FUNCTION_BLOCK FB_TopMold_OLD
VAR CONSTANT
	sCycleStateTextDef: ARRAY[0..25]  OF STRING :=	
		['State 0: Wait for Start',
		'State 1: Wait for signal to start move down',
		'State 2: Move down',
		'State 3: Drying lock time, Building pressure',
		'State 4: Start drying time',
		'State 5: Open pressure relief valve',
		'State 6: Vacuum time closed',
		'State 7: Move up',
		'State 8: Wait until take out unit is moving up and start blowoff',
		'State 9: Await blowoff time and stop blowoff',
		'State 10:',
		'State 11:',
		'State 12:',
		'State 13:',
		'State 14:',
		'State 15:',
		'State 16:',
		'State 17:',
		'State 18:',
		'State 19:',
		'State 20: Stop cycle state',																
		'State 21: Stop cycle state',
		'State 22:',
		'State 23:',
		'State 24:',
		'State 25:Stop direct state'];
	
	tCycleStateTimeouts: ARRAY[0..10] OF TIME := 
		[T#10S,T#10S,T#10S,T#10S,T#10S,T#10S,T#10S,T#10S,T#10S,T#10S,
		T#10S];

	sInitStateTextDef: ARRAY[0..10] OF STRING :=
		['State 0: Wait for Init Start',
		'State 1: Await pressure relief',
		'State 2: Move up',
		'State 3: Description Init State 3',
		'State 4: Description Init State 4',
		'State 5: Description Init State 5',
		'State 6: Description Init State 6',
		'State 7: Description Init State 7',
		'State 8: Description Init State 8',
		'State 9: Description Init State 9',
		'State 10: Stop init state'];

	tInitStateTimeouts: ARRAY[0..10] OF TIME := 
		[T#10S,T#10S,T#10S,T#10S,T#10S,T#10S,T#10S,T#10S,T#10S,T#10S
		,T#10S];
END_VAR

VAR_INPUT
	mxReset							: BOOL;	(*Reset Error*)
	mxEmergency						: BOOL;
	mxAutoMode						: BOOL; (* TRUE = Automode *)
	mxEmptyMachine					: BOOL;
	mxEnableHeating					: BOOL;

	mxResetCycleState				: BOOL;
	mxResetInitState				: BOOL;
	mxForceInit						: BOOL; (*Reset Calibration Flag*)

	mxMoveDown						: BOOL; (* Signal from bottommold *)
	mxMoveUp						: BOOL; (* Drying finished or transfer ready with new product *)
	mxTakeOutIsMovingUp: BOOL;
	RHSR_Blocked 					: BOOL;
END_VAR
VAR_IN_OUT
	MachParameters					: ST_TopMoldMachPar;
	ProdParameters					: ST_TopMoldProdPar;
END_VAR
VAR_OUTPUT
(*Errors*)
	Errors							: ST_TopMoldErrors;
	mxErrorInit						: BOOL;		(* Error, stop immediately. Initialisation neccesary *)
	mxErrorStopinPos				: BOOL;		(* Error, stop in position. Only reset neccesary *)

(* State vars *)
	mxCycleBusy						: BOOL;
	mxInitBusy						: BOOL;
	
(* Vars *)
	mxInitialized					: BOOL;
	
	mxIsUp							: BOOL;
	mxIsDown						: BOOL;
	mxCilIsMovingIn					: BOOL;
	mxCilIsMovingOut				: BOOL;
	mxCilIsIn						: BOOL;
	mxCilIsOut						: BOOL;	
END_VAR
VAR
(* State vars *)
	miCycleState					: INT :=0;
	miCycleOldstate					: INT :=0;
	mxCycleTransitionState			: BOOL := FALSE;
	sCycleStateText					: STRING;
	exCycleTimeOut					: BOOL;		(* Timeout for the whole programcycle *)
	CycleTimeout					: TON;
	CycleTimeOutUpFlank				: R_TRIG;
	mxCycleTimeoutEnable			: BOOL;
	CycleTime						: REAL;
	mxCycleHasError					: BOOL;
	miStopState						: INT;
	mxStartCycle					: BOOL;
	mxStopCycle						: BOOL;
	mxStopDirect					: BOOL;
	
	miInitState						: INT	:=0;
	miInitOldstate					: INT	:=0;
	mxInitTransitionState			: BOOL	:= FALSE;
	sInitStateText					: STRING;
	exInitTimeOut					: BOOL;		(* Timeout for the whole programcycle *)
	InitTimeout						: TON;
	InitTimeOutUpFlank				: R_TRIG;
	mxInitTimeoutEnable				: BOOL;
	InitTime						: REAL;
	mxInitHasError					: BOOL;
	mxStartInit						: BOOL;
	mxStopInit						: BOOL;
(* Objects *)
	HydraulicCilinder				: FB_HydraulicCilinderAnalog;
	Vacuum							: FB_MonoValveNoFdbck;
	BlowOff							: FB_MonoValveNoFdbck;
	HeatingZone						: ARRAY [1..6] OF FB_Heatingzone;
(* Vars *)
	T_DryingTime					: TON;
	T_BlowOffClosed					: TON;
	RT_TakeOutIsMovingUp			: R_TRIG;
	T_DryingMoldLock				: TON;
	T_VacuumTimeClosed				: TON;
	T_BlowOff						: TON;
END_VAR

Error();
Init();
Cycle();
Objects();

ACTION Cycle:
(*StateChange (Transition)  Signalgeneration*)
mxCycleTransitionState:=(miCycleState<>miCycleOldstate);
(*State text*)
sCycleStateText:=sCycleStateTextDef[miCycleState];
(*Timeout Watchdog for Statemachine*)
mxCycleTimeoutEnable:=NOT (miCycleState=0) AND NOT mxReset;

CycleTimeout(IN:=mxCycleTimeoutEnable  , PT:=tCycleStateTimeouts[miCycleState] );
CycleTimeOutUpFlank(CLK:=CycleTimeout.Q );
miCycleOldstate:=miCycleState;

(*Set Errorbit when Raising edge of Timeout has been detected*)
IF CycleTimeOutUpFlank.Q THEN
	exCycleTimeOut:=TRUE; 			(* 1 Timeout for the whole programcycle *)
END_IF

(*Function to reset the Statemachine*)
IF mxResetCycleState THEN
	mxResetCycleState:= FALSE;
	mxInitialized := FALSE;
		
	miCycleState:=0;
	miCycleOldstate:=miCycleState;
	mxCycleTransitionState:=FALSE;

	mxStartCycle:= FALSE;
	mxStopCycle:= FALSE;
	mxStopDirect:=FALSE;
	mxIsDown := FALSE;
	mxIsUp := FALSE;
	mxMoveUp := FALSE;
	mxMoveDown := FALSE;

	T_DryingTime.IN:= FALSE;
	T_DryingMoldLock.IN:= FALSE;
	T_VacuumTimeClosed.IN:= FALSE;
	T_BlowOffClosed.IN:= FALSE;
	T_BlowOff.IN:=FALSE;	
	
	HydraulicCilinder.M_Stop();
END_IF

(*Definition State has Error*)
mxCycleHasError:=FALSE;

T_DryingTime(IN:= , PT:= MachParameters.DryingTime);
T_DryingMoldLock(IN:= , PT:= MachParameters.DryingPressureLockTime);
T_VacuumTimeClosed(IN:= , PT:= MachParameters.VacuumTimeClosed);
T_BlowOffClosed(IN:= (BlowOff.mxIsOn AND (miCycleState=3 OR miCycleState=4)) AND mxAutoMode, PT:= MachParameters.BlowOffTimeClosed);
T_BlowOff(IN:=, PT:=MachParameters.BlowOffToTakeOut);

IF T_BlowOffClosed.Q THEN BlowOff.M_Off(); END_IF


(*Cycle State's*)
CASE miCycleState OF

	(* Cycle:
	LEEG beginnen
		-wacht op signaal vanuit bottommold, naar beneden
		-Naar beneden om product te drogen
		-als bijna dicht dan extra druk opbouwen
		-Na droogtijd/transfer up wait time, relief presure
		-vacuum aan, omhoog, signal to bottom mold -> vac of blow on
		-signaal Mold is up -> bottom mold
		-Wacht op bottom mold is in
		-Wacht op takeout unit is omhoog (als enabled)
		-blow off aan

	*)
	0:
		IF mxStartCycle THEN
			mxStartCycle:= FALSE;

			miCycleState:= 1;
		END_IF

	(* wait for move down *)	
	1:
		IF mxStopDirect THEN
			mxStopDirect:= FALSE;
			
			miCycleState:= 25;
		ELSIF mxStopCycle AND mxEmptyMachine THEN
			mxEmptyMachine:= FALSE;
			
			miCycleState:= 0;
		ELSIF mxStopCycle THEN
			mxStopCycle:= FALSE;
			
			miStopState:= miCycleState;
			miCycleState:= 0;
		ELSIF mxMoveDown THEN			
			mxMoveDown:= FALSE;
			mxMoveUp:= FALSE;
			
			mxIsUp:= FALSE;
			
			miCycleState:= 2;
		END_IF
		
	(* Move down *)
	2:
		IF mxStopDirect THEN
			mxStopDirect:= FALSE;

			miCycleState:= 25;(*Stop direct*)
		ELSIF mxStopCycle THEN
			mxStopCycle:= FALSE;
			
			miStopState:= miCycleState;
			miCycleState:= 20;
		ELSIF HydraulicCilinder.M_Move(EndPosition:=ProdParameters.PositionDownStop, NormalSpeed:=MachParameters.SpeedDownNormal, 
										SlowPosition:=ProdParameters.PositionDownStop + ProdParameters.PositionDownSlow, SlowSpeed:=MachParameters.SpeedDownSlow, 
										CreepPosition:=ProdParameters.PositionDownStop + ProdParameters.PositionDownCreep, CreepSpeed:=MachParameters.SpeedDownCreep) THEN
			BlowOff.M_On(); 			// Blowoff stops after delay ^ at top of cylce
			miCycleState:= 3;
		END_IF

	(* Drying Lock time, build up pressure *)
	3:
		T_DryingMoldLock.IN:= TRUE;
		
		IF mxStopDirect THEN
			mxStopDirect:= FALSE;

			miCycleState:= 25;(*Stop direct*)
		ELSIF mxStopCycle THEN
			mxStopCycle:= FALSE;
			
			miStopState:= miCycleState;
			miCycleState:= 20;
		ELSIF HydraulicCilinder.M_Move(EndPosition:=ProdParameters.PositionDownStop -50.0, NormalSpeed:=MachParameters.SpeedDownNormal,
										SlowPosition:= ProdParameters.PositionDownSlow, SlowSpeed:=MachParameters.SpeedDownSlow, 
										CreepPosition:=ProdParameters.PositionDownCreep, CreepSpeed:=MachParameters.SpeedDownCreep) OR T_DryingMoldLock.Q THEN
			HydraulicCilinder.M_Stop();
			
			T_DryingMoldLock.IN:= FALSE;
			
			mxIsDown:= TRUE;
			mxIsUp:=FALSE;
			
			miCycleState:= 4;
		END_IF
	
	(* start drying *)
	4:
		T_DryingTime(IN:= TRUE);

		IF mxStopDirect THEN
			mxStopDirect:= FALSE;

			miCycleState:= 25;(*Stop direct*)
		ELSIF mxStopCycle THEN
			mxStopCycle:= FALSE;

			miStopState:=miCycleState;
			miCycleState:= 20;

		ELSIF (mxMoveUp AND T_DryingTime.Q) THEN	// changed by bateu 20180601
			mxMoveUp:= FALSE;
			T_DryingTime(IN:= FALSE);
			
			// Switch vacuum on
			Vacuum.M_On();
			
			miCycleState:= 5;
		END_IF
		
	(* Vacuum time closed *)
	5:
		T_VacuumTimeClosed.IN:= TRUE;	
		
		IF mxStopDirect THEN
			mxStopDirect:= FALSE;

			miCycleState:= 25;(*Stop direct*)
		ELSIF mxStopCycle THEN
			mxStopCycle:= FALSE;
			
			miStopState:= miCycleState;
			miCycleState:= 20;
		ELSIF T_VacuumTimeClosed.Q THEN
			T_VacuumTimeClosed.IN:= FALSE;
			
			miCycleState:= 6;
		END_IF
		
	(* Move up *)
	6:
		IF mxStopDirect THEN
			mxStopDirect:= FALSE;

			miCycleState:= 25;(*Stop direct*)
		ELSIF mxStopCycle THEN
			mxStopCycle:= FALSE;

			miStopState:= miCycleState;
			miCycleState:= 20;
		ELSIF HydraulicCilinder.M_Move(EndPosition:= MachParameters.PositionUpStop,  NormalSpeed:= MachParameters.SpeedUpNormal, 
										SlowPosition:= MachParameters.PositionUpStop - MachParameters.PositionUpSlow, SlowSpeed:= MachParameters.SpeedUpSlow, 
										CreepPosition:=MachParameters.PositionUpStop - MachParameters.PositionUpCreep, CreepSpeed:=MachParameters.SpeedUpCreep) THEN
			mxIsUp:= TRUE;
			mxIsDown:= FALSE;
			mxMoveUp:= FALSE;
			
			miCycleState:= 7;
		END_IF
		
	(* Wait until takeout is moving up *)	
	7:
		IF mxStopDirect THEN
			mxStopDirect:= FALSE;

			miCycleState:= 25;(*Stop direct*)
		ELSIF mxStopCycle THEN
			mxStopCycle:= FALSE;
			HydraulicCilinder.M_Stop();

			miStopState:= miCycleState;
			miCycleState:= 20;
		ELSIF mxTakeOutIsMovingUp THEN
			Vacuum.M_Off();
			BlowOff.M_On();
			
			miCycleState:= 8;
		END_IF
		
	(* Await Blowoff*)	
	8:
		T_BlowOff.IN := TRUE;
	
		IF mxStopDirect THEN
			mxStopDirect:= FALSE;

			miCycleState:= 25;(*Stop direct*)
		ELSIF mxStopCycle THEN
			mxStopCycle:= FALSE;
			HydraulicCilinder.M_Stop();

			miStopState:= miCycleState;
			miCycleState:= 20;
		ELSIF T_BlowOff.Q THEN
			BlowOff.M_Off();
			
			T_BlowOff.IN := FALSE;
			miCycleState:= 1;
		END_IF

	(* Stop Cycle, wait for pressure slow setpoint reached by rebotech*)
	20:
		IF mxStopDirect THEN
			mxStopDirect:= FALSE;
			
			miCycleState:= 25;
		ELSIF TRUE THEN
 			
			miCycleState:= 21;
		END_IF

	(* Stop cycle, wait for start *)
	21:	
		IF mxStopDirect THEN
			mxStopDirect:= FALSE;

			miCycleState:= 25;
		ELSIF mxStartCycle THEN

			miCycleState:= miStopState;
		END_IF
	(* Stop Direct *)	
	25:
		mxStartCycle:= FALSE;
		mxStopCycle:= FALSE;
		mxInitialized:= FALSE;

		T_DryingTime.IN:= FALSE;
		
		HydraulicCilinder.M_StopDirect();
		Vacuum.M_Off(); (* When product do not switch off *)
		BlowOff.M_Off();
	
		miCycleState:= 0;

END_CASE

mxCycleBusy:= miCycleState<>0 AND NOT (miCycleState=21);
END_ACTION

ACTION Error:


(* ****************************************************************************** *)
mxErrorStopInPos:= HydraulicCilinder.mxErrorStopInPos;
mxErrorInit:= HydraulicCilinder.mxErrorInit
			OR HeatingZone[1].mxErrorInit
			OR HeatingZone[2].mxErrorInit
			OR HeatingZone[3].mxErrorInit
			OR HeatingZone[4].mxErrorInit
			OR HeatingZone[5].mxErrorInit
			OR HEatingZone[6].mxErrorInit;
END_ACTION

ACTION Init:
(*StateChange (Transition)  Signalgeneration*)
mxInitTransitionState:=(miInitState<>miInitOldstate);
(*State text*)
sInitStateText:=sInitStateTextDef[miInitState];
(*Timeout Watchdog for Statemachine*)
mxInitTimeoutEnable:=NOT (miInitState=0)  AND NOT mxReset;

InitTimeout(IN:=mxInitTimeoutEnable  , PT:=tInitStateTimeouts[miInitState] );
InitTimeOutUpFlank(CLK:=InitTimeout.Q );
miInitOldstate:=miInitState;

(*Set Errorbit when Raising edge of Timeout has been detected*)
IF InitTimeOutUpFlank.Q THEN
	exInitTimeOut:=TRUE; 			(* 1 Timeout for the whole programcycle *)
END_IF

(*Function to reset the Statemachine*)
IF mxResetInitState THEN
	mxResetInitState:=FALSE;
	miInitState:=0;
	miInitOldstate:=miInitState;
	mxInitTransitionState:=FALSE;
	
	mxStartInit:= FALSE;
	mxStopInit:= FALSE;		
END_IF

(*Definition State has Error*)
mxInitHasError:=FALSE;

(*Init State's*)
CASE miInitState OF
	0:
		IF mxStartInit THEN
			mxStartInit:= FALSE;
			mxInitialized:=FALSE;
			
			Vacuum.M_Off();
			BlowOff.M_Off();

			miInitState:= 1;
		END_IF
		
	(* Move Up *)	
	1:
		IF mxStopInit THEN
			mxStopInit:= FALSE;

			miInitState:= 10;	
		END_IF
		
		IF HydraulicCilinder.ActPosition > MachParameters.PositionUpStop THEN // Move down
			IF HydraulicCilinder.M_Move(EndPosition:=MachParameters.PositionUpStop, NormalSpeed:= MachParameters.SpeedUpNormal, 
											SlowPosition:=MachParameters.PositionUpStop - MachParameters.PositionUpSlow, SlowSpeed:=MachParameters.SpeedUpSlow, 
											CreepPosition:=MachParameters.PositionUpStop - MachParameters.PositionUpCreep,	CreepSpeed:=MachParameters.SpeedUpCreep ) THEN
			mxInitialized:= TRUE; (* Return val *)
			miInitState:= 0;	
			END_IF
		ELSE
			IF HydraulicCilinder.M_Move(EndPosition:=MachParameters.PositionUpStop, NormalSpeed:= MachParameters.SpeedUpNormal, 
											SlowPosition:=MachParameters.PositionUpStop + MachParameters.PositionUpSlow, SlowSpeed:=MachParameters.SpeedUpSlow, 
											CreepPosition:=MachParameters.PositionUpStop + MachParameters.PositionUpCreep,	CreepSpeed:=MachParameters.SpeedUpCreep ) THEN
			mxInitialized:= TRUE; (* Return val *)
			miInitState:= 0;	
			END_IF
		END_IF

	(* Stop Init *)
	10:
		HydraulicCilinder.M_Stop();

		mxStartInit:= FALSE;
		mxStopInit:= FALSE;
		mxInitialized:=FALSE;					

		miInitState:= 0;
END_CASE

mxInitBusy:= miInitState<>0;
END_ACTION

METHOD M_EmptyMachine

IF mxCycleBusy THEN
	mxEmptyMachine:= TRUE;	
END_IF
END_METHOD

METHOD M_StartCycle

IF NOT mxCycleBusy THEN
	mxStartCycle:= TRUE;	
	mxStopCycle := FALSE;
END_IF
END_METHOD

METHOD M_StartInit

IF NOT mxInitBusy THEN 
	mxStartInit:= TRUE; 
END_IF
END_METHOD

METHOD M_StopCycle

IF mxCycleBusy THEN 
	mxStopCycle:= TRUE; 
END_IF
END_METHOD

METHOD M_StopDirect

IF mxCycleBusy THEN
	mxStopDirect:= TRUE;	
END_IF
END_METHOD

METHOD M_StopInit

IF mxInitBusy THEN 
	mxStopInit:= TRUE; 
END_IF
END_METHOD

ACTION Objects:
(* Object Calls *)
HydraulicCilinder(
	mxReset:= mxReset, 
	mxEmergency:= mxEmergency, 
	mxAutoMode:= mxAutoMode, 
	EndPositionIn:= MachParameters.PositionUpStop,
	EndPositionOut:= ProdParameters.PositionDownStop,
	OffsetPosition:= MachParameters.PositionOffsetZero,
	OffsetAlarmPosition:= MachParameters.PositionOffsetAlarm,
	PositionPhysicalMeasured:=MachParameters.PositionPhyscialMeasured,
	PositionPhysicalMeasuredOld:=MachParameters.PositionPhysicalMeasuredOld,
	PhysicalOffsetPos:=MachParameters.PhysicalOffsetPos,
	RHSR_Blocked:=RHSR_Blocked,
	mxIsMovingIn=> mxCilIsMovingIn, 
	mxIsMovingOut=> mxCilIsMovingOut, 
	ManSpeedCreepIn:=MachParameters.SpeedUpCreep,
	ManSpeedCreepOut:=MachParameters.SpeedDownCreep,
	ManSpeedSlowIn:=MachParameters.SpeedUpSlow,
	ManSpeedSlowOut:=MachParameters.SpeedDownSlow,
	ManSpeedIn:=MachParameters.SpeedUpNormal,
	ManSpeedOut:=MachParameters.SpeedDownNormal,
	mxIsIn=> mxCilIsIn, 
	mxIsOut=> mxCilIsOut,
	Errors=> Errors.Hydraulic);
	
Vacuum(
	mxReset:= mxReset, 
	mxEmergency:= mxEmergency, 
	mxAutoMode:= mxAutoMode);
	
BlowOff(
	mxReset:= mxReset, 
	mxEmergency:= mxEmergency, 
	mxAutoMode:= mxAutoMode);


HeatingZone[1](
	mxReset:= mxReset,
	mxEmergency:=mxEmergency,
	mxEnableHeating:=mxEnableHeating,
	MachParameters:=MachParameters.HeatingZone[1],
	Errors=> Errors.HeatingZone[1]);
	
HeatingZone[2](
	mxReset:= mxReset,
	mxEmergency:=mxEmergency,
	mxEnableHeating:=mxEnableHeating,
	MachParameters:=MachParameters.HeatingZone[2],
	Errors=> Errors.HeatingZone[2]);

HeatingZone[3](
	mxReset:= mxReset,
	mxEmergency:=mxEmergency,
	mxEnableHeating:=mxEnableHeating,
	MachParameters:=MachParameters.HeatingZone[3],
	Errors=> Errors.HeatingZone[3]);

HeatingZone[4](
	mxReset:= mxReset,
	mxEmergency:=mxEmergency,
	mxEnableHeating:=mxEnableHeating,
	MachParameters:=MachParameters.HeatingZone[4],
	Errors=> Errors.HeatingZone[4]);

HeatingZone[5](
	mxReset:= mxReset,
	mxEmergency:=mxEmergency,
	mxEnableHeating:=mxEnableHeating,
	MachParameters:=MachParameters.HeatingZone[5],
	Errors=> Errors.HeatingZone[5]);

HeatingZone[6](
	mxReset:= mxReset,
	mxEmergency:=mxEmergency,
	mxEnableHeating:=mxEnableHeating,
	MachParameters:=MachParameters.HeatingZone[6],
	Errors=> Errors.HeatingZone[6]);
END_ACTION

END_FUNCTION_BLOCK

(* stored: Version 1.1.0.1, ProductVersion 3.1.4020.12
   POU FB_TopMold_OLD: Id {12607023-8663-43a6-a062-ab85428ca54a}, SpecialFunc None
   Action Cycle: Id {efc7c7f2-e575-432e-8f92-c0d983c8a7bd}
   Action Error: Id {9fed989a-c5f4-4e97-8346-93c202e80970}
   Action Init: Id {00dcca80-6985-4b0f-9286-e5ff5cf89d17}
   Method M_EmptyMachine: Id {27910021-41c1-4a63-8ba3-ec2f3208a183}
   Method M_StartCycle: Id {b74b68d9-0a5f-44e0-b923-7dde95c117fe}
   Method M_StartInit: Id {6e24aad9-3dfe-424b-9b9b-15513f156b44}
   Method M_StopCycle: Id {bd8eaf1e-a3dc-4bac-8bf2-bc889cce4463}
   Method M_StopDirect: Id {83dfc892-7419-4c1e-a6f1-1efe211cc35f}
   Method M_StopInit: Id {a96f3438-9240-4c23-bedd-9a4ca9fa6371}
   Action Objects: Id {564e1988-4c27-4b84-b369-8a44ad57ddd9} *)
